FUNCTION_BLOCK FB_SL3K4
VAR
    stTopBlade : REFERENCE TO ST_MotionStage;
    stBottomBlade : REFERENCE TO ST_MotionStage;
    stNorthBlade : REFERENCE TO ST_MotionStage;
    stSouthBlade : REFERENCE TO ST_MotionStage;

    fbFFHWO       : REFERENCE TO FB_HardwareFFOutput;   // Fast Fault hardware relay IO (passed in)
    fbArbiter     : REFERENCE TO FB_Arbiter;            // PMPS Arbiter block (passed in)
    fbPerMotorFFO: FB_PerMotorFFOND;
    fbEncErrorFFO: FB_EncErrorFFO;
    ffProgErr    : FB_FastFault;
    {attribute 'pytmc' := 'pv: STATE'}
    stEpicsToPlc     : ST_StateEpicsToPlc;
    {attribute 'pytmc' := 'pv: STATE'}
    stPMPSEpicsToPlc : ST_StatePMPSEpicsToPlc;


	(* Axis X1 *)
	{attribute 'TcLinkToOSO' := '
		.stDS402Drive.nModeOfOperationNC      := <0,8,0>TINC^NC-Task 1^Axes^M13_DREAM_SLIT_MMT_X1^Drive^Outputs^Out^nCtrl5;
		.stDS402Drive.nDS402DriveControlNC.0  := <0,8,0>TINC^NC-Task 1^Axes^M13_DREAM_SLIT_MMT_X1^Drive^Outputs^Out^nCtrl1;
		.stDS402Drive.nDS402DriveControlNC.1  := <8,8,0>TINC^NC-Task 1^Axes^M13_DREAM_SLIT_MMT_X1^Drive^Outputs^Out^nCtrl2;
	'}
	{attribute 'TcLinkTo' := '
		.stDS402Drive.nSlaveAddr              := TIID^Device 1 (EtherCAT)^TMO-DREAM-SMARACT-04^InfoData^AdsAddr^port;
		.stDS402Drive.stDS402DriveStatus      := TIID^Device 1 (EtherCAT)^TMO-DREAM-SMARACT-04^DREAM:SLIT:MMT:X1^mode/status/pos/fError TxPDO^Status Word;
		.stDS402Drive.nFollowingError         := TIID^Device 1 (EtherCAT)^TMO-DREAM-SMARACT-04^DREAM:SLIT:MMT:X1^mode/status/pos/fError TxPDO^Following Error Actual Value;
		.stDS402Drive.nModeOfOperation        := TIID^Device 1 (EtherCAT)^TMO-DREAM-SMARACT-04^DREAM:SLIT:MMT:X1^ctl/mode/pos RxPDO^Modes of Operation;
		.stDS402Drive.nModeOfOperationDisplay := TIID^Device 1 (EtherCAT)^TMO-DREAM-SMARACT-04^DREAM:SLIT:MMT:X1^mode/status/pos/fError TxPDO^Modes of Operation Display;
		.stDS402Drive.nDS402DriveControl      := TIID^Device 1 (EtherCAT)^TMO-DREAM-SMARACT-04^DREAM:SLIT:MMT:X1^ctl/mode/pos RxPDO^Control Word;
	'}
	fb_SLIT_X1 : FB_MotionStageMCS2(stPiezoStage:=Main.M13, eModule:=E_Module.CHAN2);
	
	(* Axis X2 *)
	{attribute 'TcLinkToOSO' := '
		.stDS402Drive.nModeOfOperationNC      := <0,8,0>TINC^NC-Task 1^Axes^M14_DREAM_SLIT_MMT_X2^Drive^Outputs^Out^nCtrl5;
		.stDS402Drive.nDS402DriveControlNC.0  := <0,8,0>TINC^NC-Task 1^Axes^M14_DREAM_SLIT_MMT_X2^Drive^Outputs^Out^nCtrl1;
		.stDS402Drive.nDS402DriveControlNC.1  := <8,8,0>TINC^NC-Task 1^Axes^M14_DREAM_SLIT_MMT_X2^Drive^Outputs^Out^nCtrl2;
	'}
	{attribute 'TcLinkTo' := '
		.stDS402Drive.nSlaveAddr              := TIID^Device 1 (EtherCAT)^TMO-DREAM-SMARACT-04^InfoData^AdsAddr^port;
		.stDS402Drive.stDS402DriveStatus      := TIID^Device 1 (EtherCAT)^TMO-DREAM-SMARACT-04^DREAM:SLIT:MMT:X2^mode/status/pos/fError TxPDO^Status Word;
		.stDS402Drive.nFollowingError         := TIID^Device 1 (EtherCAT)^TMO-DREAM-SMARACT-04^DREAM:SLIT:MMT:X2^mode/status/pos/fError TxPDO^Following Error Actual Value;
		.stDS402Drive.nModeOfOperation        := TIID^Device 1 (EtherCAT)^TMO-DREAM-SMARACT-04^DREAM:SLIT:MMT:X2^ctl/mode/pos RxPDO^Modes of Operation;
		.stDS402Drive.nModeOfOperationDisplay := TIID^Device 1 (EtherCAT)^TMO-DREAM-SMARACT-04^DREAM:SLIT:MMT:X2^mode/status/pos/fError TxPDO^Modes of Operation Display;
		.stDS402Drive.nDS402DriveControl      := TIID^Device 1 (EtherCAT)^TMO-DREAM-SMARACT-04^DREAM:SLIT:MMT:X2^ctl/mode/pos RxPDO^Control Word;
	'}
	fb_SLIT_X2 : FB_MotionStageMCS2(stPiezoStage:=Main.M14, eModule:=E_Module.CHAN3);
	
	(* Axis Y1 *)
	{attribute 'TcLinkToOSO' := '
		.stDS402Drive.nModeOfOperationNC      := <0,8,0>TINC^NC-Task 1^Axes^M15_DREAM_SLIT_MMT_Y1^Drive^Outputs^Out^nCtrl5;
		.stDS402Drive.nDS402DriveControlNC.0  := <0,8,0>TINC^NC-Task 1^Axes^M15_DREAM_SLIT_MMT_Y1^Drive^Outputs^Out^nCtrl1;
		.stDS402Drive.nDS402DriveControlNC.1  := <8,8,0>TINC^NC-Task 1^Axes^M15_DREAM_SLIT_MMT_Y1^Drive^Outputs^Out^nCtrl2;
	'}
	{attribute 'TcLinkTo' := '
		.stDS402Drive.nSlaveAddr              := TIID^Device 1 (EtherCAT)^TMO-DREAM-SMARACT-05^InfoData^AdsAddr^port;
		.stDS402Drive.stDS402DriveStatus      := TIID^Device 1 (EtherCAT)^TMO-DREAM-SMARACT-05^DREAM:SLIT:MMT:Y1^mode/status/pos/fError TxPDO^Status Word;
		.stDS402Drive.nFollowingError         := TIID^Device 1 (EtherCAT)^TMO-DREAM-SMARACT-05^DREAM:SLIT:MMT:Y1^mode/status/pos/fError TxPDO^Following Error Actual Value;
		.stDS402Drive.nModeOfOperation        := TIID^Device 1 (EtherCAT)^TMO-DREAM-SMARACT-05^DREAM:SLIT:MMT:Y1^ctl/mode/pos RxPDO^Modes of Operation;
		.stDS402Drive.nModeOfOperationDisplay := TIID^Device 1 (EtherCAT)^TMO-DREAM-SMARACT-05^DREAM:SLIT:MMT:Y1^mode/status/pos/fError TxPDO^Modes of Operation Display;
		.stDS402Drive.nDS402DriveControl      := TIID^Device 1 (EtherCAT)^TMO-DREAM-SMARACT-05^DREAM:SLIT:MMT:Y1^ctl/mode/pos RxPDO^Control Word;
	'}
	fb_SLIT_Y1 : FB_MotionStageMCS2(stPiezoStage:=Main.M15, eModule:=E_Module.CHAN1);
	
	(* Axis Y2 *)
	{attribute 'TcLinkToOSO' := '
		.stDS402Drive.nModeOfOperationNC      := <0,8,0>TINC^NC-Task 1^Axes^M16_DREAM_SLIT_MMT_Y2^Drive^Outputs^Out^nCtrl5;
		.stDS402Drive.nDS402DriveControlNC.0  := <0,8,0>TINC^NC-Task 1^Axes^M16_DREAM_SLIT_MMT_Y2^Drive^Outputs^Out^nCtrl1;
		.stDS402Drive.nDS402DriveControlNC.1  := <8,8,0>TINC^NC-Task 1^Axes^M16_DREAM_SLIT_MMT_Y2^Drive^Outputs^Out^nCtrl2;
	'}
	{attribute 'TcLinkTo' := '
		.stDS402Drive.nSlaveAddr              := TIID^Device 1 (EtherCAT)^TMO-DREAM-SMARACT-05^InfoData^AdsAddr^port;
		.stDS402Drive.stDS402DriveStatus      := TIID^Device 1 (EtherCAT)^TMO-DREAM-SMARACT-05^DREAM:SLIT:MMT:Y2^mode/status/pos/fError TxPDO^Status Word;
		.stDS402Drive.nFollowingError         := TIID^Device 1 (EtherCAT)^TMO-DREAM-SMARACT-05^DREAM:SLIT:MMT:Y2^mode/status/pos/fError TxPDO^Following Error Actual Value;
		.stDS402Drive.nModeOfOperation        := TIID^Device 1 (EtherCAT)^TMO-DREAM-SMARACT-05^DREAM:SLIT:MMT:Y2^ctl/mode/pos RxPDO^Modes of Operation;
		.stDS402Drive.nModeOfOperationDisplay := TIID^Device 1 (EtherCAT)^TMO-DREAM-SMARACT-05^DREAM:SLIT:MMT:Y2^mode/status/pos/fError TxPDO^Modes of Operation Display;
		.stDS402Drive.nDS402DriveControl      := TIID^Device 1 (EtherCAT)^TMO-DREAM-SMARACT-05^DREAM:SLIT:MMT:Y2^ctl/mode/pos RxPDO^Control Word;
	'}
	fb_SLIT_Y2 : FB_MotionStageMCS2(stPiezoStage:=Main.M16, eModule:=E_Module.CHAN2);

 	{attribute 'pytmc' := 'pv: SL3K4:STATE'}
    eSL3K4State           : E_SL3K4STATE;

    astMotionStage      : ARRAY[1..4] OF  ST_MotionStage;


    // PMPS parameter sets (setup at config time)
    MaintenanceParams    : ST_BeamParams := PMPS_GVL.cst0RateBeam;
    NormalParams         : ST_BeamParams := PMPS_GVL.cst0RateBeam;
    nUID_Maint           : UDINT := 1001;
    nUID_Norm            : UDINT := 1000;
    nActiveMotorCount    : UINT := 4;

    // Status
    abBladeEnable        : ARRAY[1..4] OF BOOL;
    bSafeToMove          : BOOL;
    bLocked              : BOOL;
    bMaintenanceActive   : BOOL;
    bFastFault           : BOOL;
    bEncoderFault        : BOOL;
    bPMPSAllowed         : BOOL;
    bPMPSMaintenance     : BOOL;
    bProgrammerError     : BOOL;
    sStatusMsg           : STRING;

    // Internal logic
    allAxesIdle   : BOOL;
    anyAxisError  : BOOL;
    bModeChange   : BOOL;
    bArbiterError : BOOL;
    nPrevMode     : E_SL3K4State := E_SL3K4State.NORMAL; // Track last asserted state to manage assertions
    axis          : INT;
	// SL3K4 Beam parameters
	sDeviceName : STRING := 'SL3K4';
    astSl3k4State : ARRAY[1..2] OF ST_SL3K4State;
	// get PMPDB state parameters
    fbSL3K4ReadPMPSDB	: FB_SL3K4ReadPMPSDB(astSl3k4State:=astSl3k4State, fbFFHWO:= GVL_PMPS.fbFastFaultOutput1);
END_VAR

// --- Assign blade references each scan ---
astMotionStage[1] := stTopBlade;
astMotionStage[2] := stBottomBlade;
astMotionStage[3] := stNorthBlade;
astMotionStage[4] := stSouthBlade;

// --- Mode logic
bMaintenanceActive := (eSL3K4State = E_SL3K4STATE.MAINTENANCE);

// --- Remove previous arbiter request if mode has changed
IF nPrevMode <>  eSL3K4State THEN
    IF nPrevMode = E_SL3K4STATE.NORMAL THEN
        fbArbiter.RemoveRequest(nUID_Norm);
    ELSIF nPrevMode = E_SL3K4STATE.MAINTENANCE THEN
        fbArbiter.RemoveRequest(nUID_Maint);
    END_IF
    nPrevMode :=  eSL3K4State;
END_IF

// --- Add current PMPS request (duplicate-protected, maintenance or normal)
IF bMaintenanceActive THEN
    IF NOT fbArbiter.CheckRequest(nUID_Maint) THEN
        fbArbiter.AddRequest(
			nReqID := nUID_Maint, 
			sDevName:=sDeviceName, 
			stReqBP := astSl3k4State[E_SL3K4State.MAINTENANCE].stPMPS.stBeamParams,
		);
    END_IF
    bPMPSMaintenance := fbArbiter.CheckRequest(nUID_Maint);
ELSE
    IF NOT fbArbiter.CheckRequest(nUID_Norm) THEN
        fbArbiter.AddRequest(
			nReqID := nUID_Norm, 
			sDevName:=sDeviceName, 
			stReqBP := astSl3k4State[E_SL3K4State.NORMAL].stPMPS.stBeamParams,
		);
    END_IF
    bPMPSAllowed := fbArbiter.CheckRequest(nUID_Norm);
END_IF

bArbiterError := fbArbiter.bFault OR fbArbiter.ArbitrationDenied;

allAxesIdle := TRUE;
anyAxisError := FALSE;
FOR axis := 1 TO 4 DO
    IF astMotionStage[axis].bBusy THEN allAxesIdle := FALSE; END_IF
    IF astMotionStage[axis].bFault THEN anyAxisError := TRUE; END_IF
END_FOR

// ---- Manual/Scatter logic for axis enable/locking ----
FOR axis := 1 TO 4 DO
    IF bMaintenanceActive AND bPMPSMaintenance AND NOT bArbiterError THEN
        astMotionStage[axis].bPowerSelf   := TRUE;  // Scatter block is "owner"
        astMotionStage[axis].bAllEnable   := bEnableMotion;
        astMotionStage[axis].bHardwareEnable := TRUE;
        astMotionStage[axis].nBrakeMode   := ENUM_StageBrakeMode.NO_BRAKE;
        abBladeEnable[axis] := astMotionStage[axis].bAllEnable;
    ELSE
        astMotionStage[axis].bPowerSelf   := FALSE;
        astMotionStage[axis].bAllEnable   := FALSE;
        astMotionStage[axis].bHardwareEnable := TRUE;
        astMotionStage[axis].nBrakeMode   := ENUM_StageBrakeMode.NO_BRAKE;
        abBladeEnable[axis] := FALSE;
    END_IF
END_FOR

bSafeToMove := bMaintenanceActive AND bPMPSMaintenance AND NOT anyAxisError AND NOT bArbiterError;
bLocked := NOT bSafeToMove OR bArbiterError;

// --- Per-motor fast fault logic (uses all blades) ---
fbPerMotorFFO(
    astMotionStage := ,
    fbFFHWO := fbFFHWO,
    nActiveMotorCount := 4,
    sDeviceName := sDeviceName
);
bFastFault := fbPerMotorFFO.bFault;

// --- Encoder error fast fault (optional, if you want per-blade encoder safety) ---
fbEncErrorFFO(
    astMotionStage := [stTopBlade, stBottomBlade, stNorthBlade, stSouthBlade],
    fbFFHWO := fbFFHWO
);
bEncoderFault := fbEncErrorFFO.bFault;

// --- Programmer error: not exactly 4 axes present
bProgrammerError := nActiveMotorCount <> 4;
ffProgErr(
    i_xOK := NOT bProgrammerError,
    i_xAutoReset := TRUE,
    i_DevName := sDeviceName,
    i_Desc := 'Programmer error picking motor count',
    i_TypeCode := E_MotionFFType.INTERNAL_ERROR,
    io_fbFFHWO := fbFFHWO
);

// --- Compose status message for debug/diagnostics
IF bArbiterError THEN
    sStatusMsg := 'Arbiter error or beam permission denied.';
ELSIF bFastFault OR bEncoderFault OR bProgrammerError THEN
    sStatusMsg := 'Device fast faulted (axis, encoder, or config error)';
ELSIF bMaintenanceActive THEN
    sStatusMsg := 'Maintenance: PMPS safe, axes enabled for manual scatter/homing.';
ELSE
    sStatusMsg := 'Normal: Axes locked for PMPS protection.';
END_IF

//FB_Init is always available implicitly and it is used primarily for initialization.
//The return value is not evaluated. For a specific influence, you can also declare the
//methods explicitly and provide additional code there with the standard initialization
//code. You can evaluate the return value.
METHOD FB_Init: BOOL
VAR_INPUT
    bInitRetains: BOOL; // TRUE: the retain variables are initialized (reset warm / reset cold)
    bInCopyCode: BOOL;  // TRUE: the instance will be copied to the copy code afterward (online change)  

    stRefX1  : REFERENCE TO ST_MotionStage;
    stRefX2	: REFERENCE TO ST_MotionStage;
    stRefY1  : REFERENCE TO ST_MotionStage;
    stRefY2  : REFERENCE TO ST_MotionStage;
    fbRefFFHWO       : REFERENCE TO FB_HardwareFFOutput;   // Fast Fault hardware relay IO (passed in)
    fbRefArbiter     : REFERENCE TO FB_Arbiter;            // PMPS Arbiter block (passed in)
END_VAR
THIS^.stRefX1 := stRefX1;
THIS^.stRefX2 := stRefX2;
THIS^.stRefY1 := stRefY1;
THIS^.stRefY2 := stRefY2;

THIS^.fbRefFFHWO       := fbRefFFHWO;   
THIS^.fbRefArbiter     := fbRefArbiter;
END_METHOD

END_FUNCTION_BLOCK

(* stored: Version 1.1.0.1
   POU FB_SL3K4: Id {dec1d628-e499-461c-bd3b-fc39c76517dd}, SpecialFunc None
   Method FB_Init: Id {69f5868f-3054-4962-be93-290684220d71} *)
